{attribute 'qualified_only'}
VAR_GLOBAL
	//HMI Stuff
	HMI_OUT_Digital 	: ARRAY[0..20] OF BOOL;
	HMI_OUT_Analog 		: ARRAY[0..10] OF INT;
	
	HMI_IN_Digital 		: ARRAY[0..10] OF BOOL;
	HMI_IN_Analog 		: ARRAY[0..20] OF INT;
	
	HMI_IN_Temp 		: ARRAY[0..4] OF REAL;
	
	HMI_State			: INT;
	
	fbGetLocalSystemTime: FB_LocalSystemTime;
	sSystemDateTime : STRING;
	sSystemTime		: STRING;
	sSystemDate		: STRING;
	
	HMI_ArrayGraph1 : ARRAY[0..1] OF INT;
	HMI_ArrayGraph2 : ARRAY[0..1] OF INT;
	HMI_ArrayGraph3 : ARRAY[0..1] OF INT;
	
END_VAR

(* stored: Version 1.1.0.1, ProductVersion 3.1.4024.12
   GVL HMI_Global: Id {4c665789-2eb9-425e-8cec-ee37673d3e12} *)
